(* PLC project PID, Beckhoff Automation GmbH TwinCAT PLC Control 3.5.13.21 *)
(* stored: creationDateTime 2022-05-17T15:59:35.6785638, modificationDateTime 2022-05-17T15:59:35.6785638 *)

TYPE S_PID_Param :
STRUCT
	Kp		: REAL;		// Reglerverstaerkung
	Ti		: REAL;		// I Anteil
	Td 		: REAL; 	// D Anteil
	N		: UINT;		// D-Anteil Filterung
	Tr		: REAL;		// Weight of Anti reset windup back calculation
	ARW		: BOOL;		// Anti reset Windup aktiv
	umin	: REAL;		// Steuergroesse minimaler Wert
	umax	: REAL;		// Steuergroesse maximaler Wert
END_STRUCT
END_TYPE
